# EPICS substitutions: iocs/mcf01/ppmacApp/pmc/xf27idf-mcf01-plc05-cpu.substitutions
file "PLC_cpu_load.pmc" { pattern {PLC} {5} }
